// Project-owned release engineering for the pneumatic press, authored in LADDER.
//
// This is an O2 DEMONSTRATION IN THE BENCH, not a per-project pattern. Core
// §6.8/§7.2 permit a sequence or an interlock to be authored in ST, SFC or LD,
// and the only way that claim is testable is to carry a rendition and compile
// it. Two renditions of one interlock is duplication §1.1 O9 would otherwise
// forbid outright - it is justified here, and ONLY here, because demonstrating
// the language choice IS this project's purpose, exactly as the three AUTO
// chain renditions are. A real project writes this once, in one language.
// FB_PressDemoUnit.RELEASE_LANGUAGE selects which one is evaluated.
//
// Same public surface as FB_PressDemoRelease so the Unit binds either without
// any other difference, and like it this is not a Fraktal module: it exposes
// named condition state and fills the Unit's authoritative release reports
// without adding an OPC UA tree node.
FUNCTION_BLOCK FB_LD_PressDemoRelease EXTENDS FB_PressDemoReleaseState
VAR
    _ramExtendOk : BOOL;
    _ramExtendKey : STRING(255);
    // AppendFailed returns the new report count. ST may discard a return value;
    // a rung has to land it somewhere, and the ENO slot is not that somewhere.
    _appendCount : INT;
END_VAR

; // Evaluated explicitly by the owning Unit after child cyclic status is available.

METHOD Setup : BOOL
VAR_INPUT
    UnitPath : STRING(255);
END_VAR
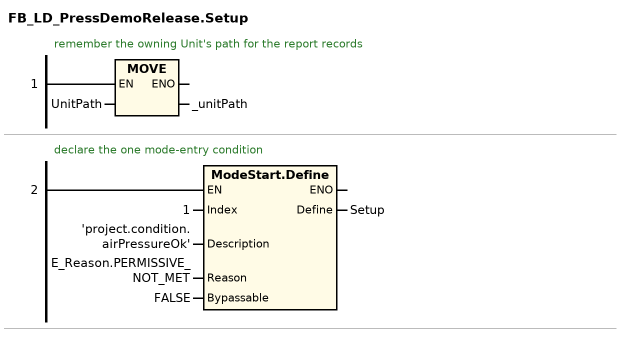
// NETWORK 1
// remember the owning Unit's path for the report records
_unitPath := UnitPath;

// NETWORK 2
// declare the one mode-entry condition
Setup := ModeStart.Define(Index := 1, Description := 'project.condition.airPressureOk', Reason := E_Reason.PERMISSIVE_NOT_MET, Bypassable := FALSE);
END_METHOD

METHOD M_Evaluate
VAR_INPUT
    PressRam : REFERENCE TO FB_CylinderCM;
    Door : REFERENCE TO FB_CylinderCM;
    PartSlide : REFERENCE TO FB_CylinderCM;
    TwoHand : REFERENCE TO FB_TwoHandStartCM;
    PneumaticPower : REFERENCE TO FB_PowerGroupCM;
    AirPressure : REFERENCE TO FB_AirPressureMonitorCM;
END_VAR
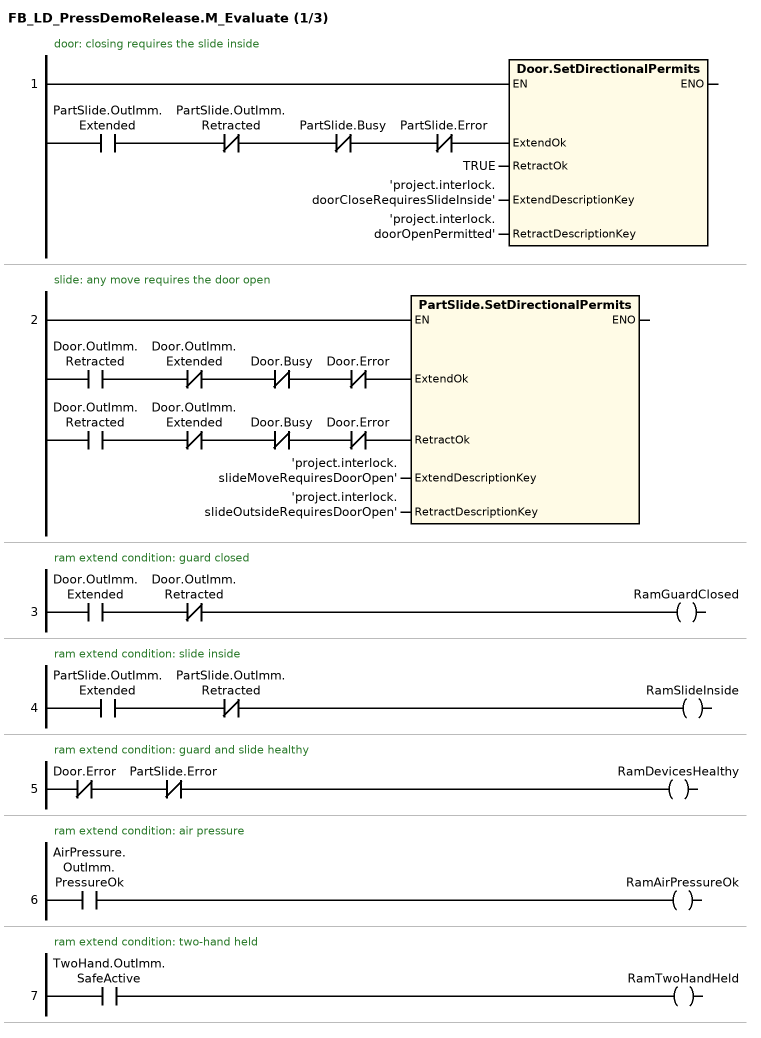
// NETWORK 1
// door: closing requires the slide inside
Door.SetDirectionalPermits(ExtendOk := PartSlide.OutImm.Extended AND NOT PartSlide.OutImm.Retracted AND NOT PartSlide.Busy AND NOT PartSlide.Error, RetractOk := TRUE, ExtendDescriptionKey := 'project.interlock.doorCloseRequiresSlideInside', RetractDescriptionKey := 'project.interlock.doorOpenPermitted');

// NETWORK 2
// slide: any move requires the door open
PartSlide.SetDirectionalPermits(ExtendOk := Door.OutImm.Retracted AND NOT Door.OutImm.Extended AND NOT Door.Busy AND NOT Door.Error, RetractOk := Door.OutImm.Retracted AND NOT Door.OutImm.Extended AND NOT Door.Busy AND NOT Door.Error, ExtendDescriptionKey := 'project.interlock.slideMoveRequiresDoorOpen', RetractDescriptionKey := 'project.interlock.slideOutsideRequiresDoorOpen');

// NETWORK 3
// ram extend condition: guard closed
RamGuardClosed := Door.OutImm.Extended AND NOT Door.OutImm.Retracted;

// NETWORK 4
// ram extend condition: slide inside
RamSlideInside := PartSlide.OutImm.Extended AND NOT PartSlide.OutImm.Retracted;

// NETWORK 5
// ram extend condition: guard and slide healthy
RamDevicesHealthy := NOT Door.Error AND NOT PartSlide.Error;

// NETWORK 6
// ram extend condition: air pressure
RamAirPressureOk := AirPressure.OutImm.PressureOk;

// NETWORK 7
// ram extend condition: two-hand held
RamTwoHandHeld := TwoHand.OutImm.SafeActive;

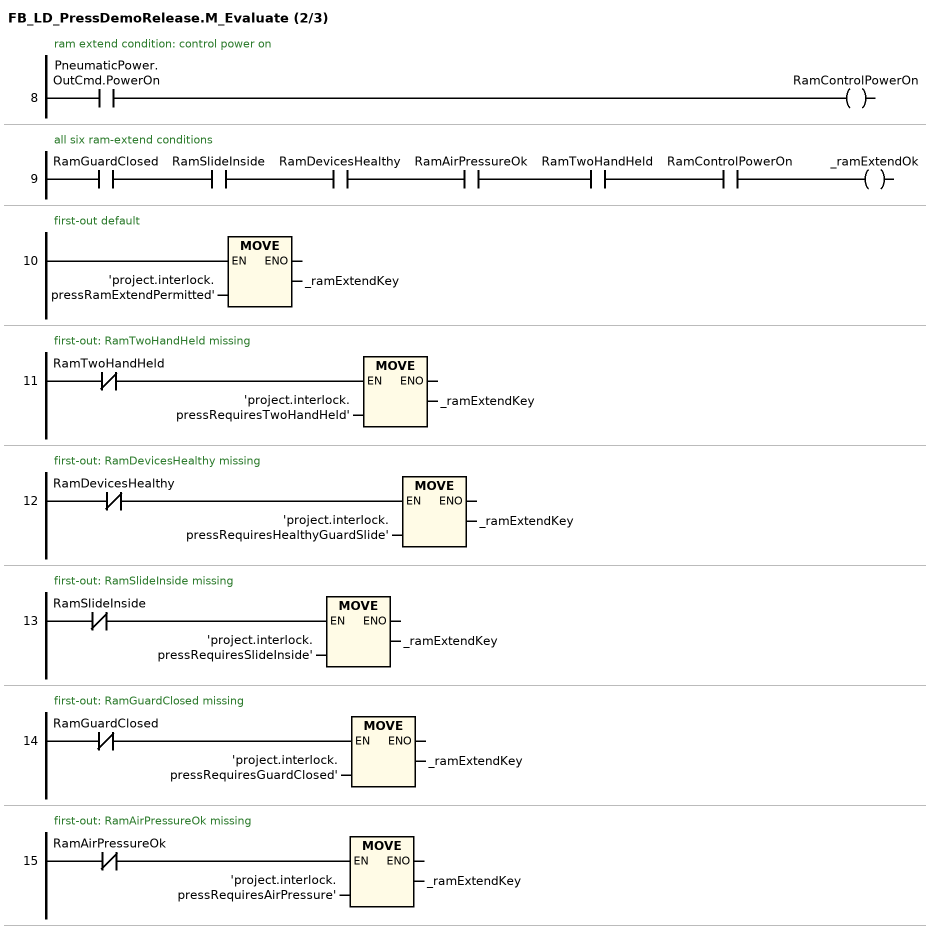
// NETWORK 8
// ram extend condition: control power on
RamControlPowerOn := PneumaticPower.OutCmd.PowerOn;

// NETWORK 9
// all six ram-extend conditions
_ramExtendOk := RamGuardClosed AND RamSlideInside AND RamDevicesHealthy AND RamAirPressureOk AND RamTwoHandHeld AND RamControlPowerOn;

// NETWORK 10
// first-out default
_ramExtendKey := 'project.interlock.pressRamExtendPermitted';

// NETWORK 11
// first-out: RamTwoHandHeld missing
IF NOT RamTwoHandHeld THEN _ramExtendKey := 'project.interlock.pressRequiresTwoHandHeld'; END_IF

// NETWORK 12
// first-out: RamDevicesHealthy missing
IF NOT RamDevicesHealthy THEN _ramExtendKey := 'project.interlock.pressRequiresHealthyGuardSlide'; END_IF

// NETWORK 13
// first-out: RamSlideInside missing
IF NOT RamSlideInside THEN _ramExtendKey := 'project.interlock.pressRequiresSlideInside'; END_IF

// NETWORK 14
// first-out: RamGuardClosed missing
IF NOT RamGuardClosed THEN _ramExtendKey := 'project.interlock.pressRequiresGuardClosed'; END_IF

// NETWORK 15
// first-out: RamAirPressureOk missing
IF NOT RamAirPressureOk THEN _ramExtendKey := 'project.interlock.pressRequiresAirPressure'; END_IF

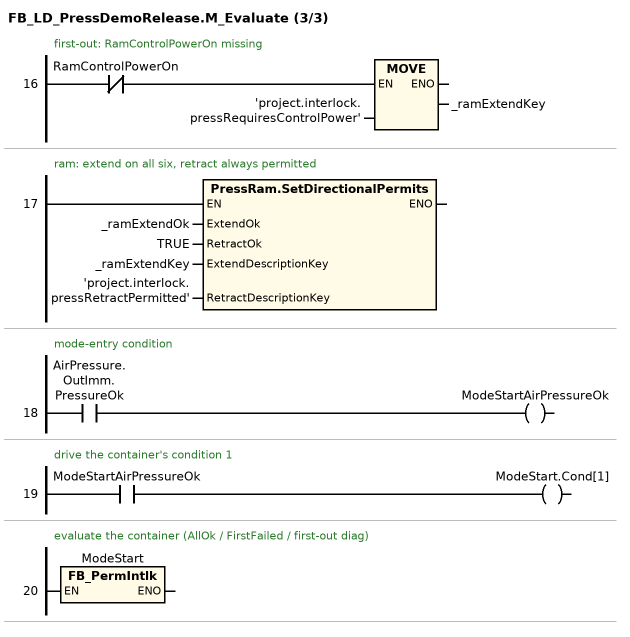
// NETWORK 16
// first-out: RamControlPowerOn missing
IF NOT RamControlPowerOn THEN _ramExtendKey := 'project.interlock.pressRequiresControlPower'; END_IF

// NETWORK 17
// ram: extend on all six, retract always permitted
PressRam.SetDirectionalPermits(ExtendOk := _ramExtendOk, RetractOk := TRUE, ExtendDescriptionKey := _ramExtendKey, RetractDescriptionKey := 'project.interlock.pressRetractPermitted');

// NETWORK 18
// mode-entry condition
ModeStartAirPressureOk := AirPressure.OutImm.PressureOk;

// NETWORK 19
// drive the container's condition 1
ModeStart.Cond[1] := ModeStartAirPressureOk;

// NETWORK 20
// evaluate the container (AllOk / FirstFailed / first-out diag)
ModeStart(); // FB_PermIntlk
END_METHOD

METHOD M_AppendStart
VAR_IN_OUT
    Report : ST_ReleaseReport;
END_VAR
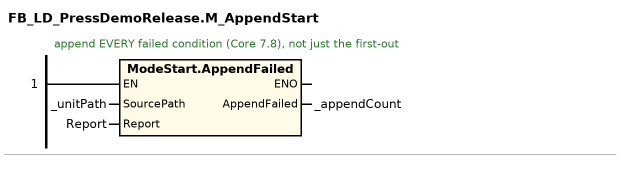
// NETWORK 1
// append EVERY failed condition (Core 7.8), not just the first-out
_appendCount := ModeStart.AppendFailed(SourcePath := _unitPath, Report := Report);
END_METHOD

// Deliberately ST, in a POU whose interlocks are ladder. This method is TARGET
// DISPATCH and bounded-report bookkeeping - matching a path against three child
// names and, failing that, writing five fields of one report row. None of that
// is condition logic, which is what O2's choice of language is about, and a
// ladder rendition of it would be longer, harder to read and no more
// demonstrative. Per-method language choice is exactly what TwinCAT offers.
METHOD M_AppendManual
VAR_INPUT
    TargetPath : STRING(255);
    Value : DINT;
    PressRam : REFERENCE TO FB_CylinderCM;
    Door : REFERENCE TO FB_CylinderCM;
    PartSlide : REFERENCE TO FB_CylinderCM;
END_VAR
VAR_IN_OUT
    Report : ST_ReleaseReport;
END_VAR
IF TargetPath = PressRam.Name THEN
    PressRam.AppendDirectionalRelease(Value := Value, Report := Report);
ELSIF TargetPath = Door.Name THEN
    Door.AppendDirectionalRelease(Value := Value, Report := Report);
ELSIF TargetPath = PartSlide.Name THEN
    PartSlide.AppendDirectionalRelease(Value := Value, Report := Report);
ELSE
    IF Report.Count < PL_Fraktal.MAX_RELEASE_REASONS THEN
        Report.Count := Report.Count + 1;
        Report.Reasons[Report.Count].Description := 'std.error.unsupportedManualTarget';
        Report.Reasons[Report.Count].ReasonCode := E_Reason.UNSUPPORTED_COMMAND;
        Report.Reasons[Report.Count].SourcePath := _unitPath;
        Report.Reasons[Report.Count].Kind := E_ReleaseKind.OTHER;
        Report.Reasons[Report.Count].Bypassable := FALSE;
    ELSE
        ; // bounded report is full; no array write is attempted
    END_IF
END_IF
END_METHOD

END_FUNCTION_BLOCK

(* stored: Version 1.1.0.1, ProductVersion 3.1.4024.12
   POU FB_LD_PressDemoRelease: Id {6b17f0c4-4d29-4b8e-9c31-2e5a7d40b911}, SpecialFunc None
   Method Setup: Id {6b17f0c4-4d29-4b8e-9c31-2e5a7d40b912}
   Method M_Evaluate: Id {6b17f0c4-4d29-4b8e-9c31-2e5a7d40b913}
   Method M_AppendStart: Id {6b17f0c4-4d29-4b8e-9c31-2e5a7d40b914}
   Method M_AppendManual: Id {6b17f0c4-4d29-4b8e-9c31-2e5a7d40b915} *)
